(* IEC 61131-3 sources: Industry-PLC-LLM/data/PLCBEAD_repo/PLCBEAD_PLCEmbed-main/PLC-BEAD/Source/GEB/DWORD_TO_TIME, 1 file *)

(* ---- DWORD_TO_TIME.ST ---- *)
FUNCTION DWORD_TO_TIME2:TIME
	VAR_INPUT
		X :	DWORD;
	END_VAR
	DWORD_TO_TIME2 := DINT_TO_TIME(DWORD_TO_DINT(X));
END_FUNCTION

PROGRAM program0
  VAR
    LocalVar0 : DWORD;
	  LocalOUT  : TIME;
  END_VAR
  	LocalOUT := DWORD_TO_TIME2(LocalVar0);
END_PROGRAM
